# EPICS autosave request: iocBoot/ioc13Raman_ps1/auto_settings.req
file "prosilica_settings.req",      P=$(P),  R=cam1:
file "NDStdArrays_settings.req",    P=$(P),  R=image1:
file "commonPlugin_settings.req",   P=$(P)
